(* Logix 5000 project; controller EuniceF_ICA14 vendor 1 type 14 code 150 rev 37.11; software revision 37.00 *)

TASK MainTask (continuous, watchdog 500 ms) : MainProgram

MODULES
   Local : vendor 1 type 14 code 150 (Compact 0, rev 37.11)
      Discrete_IO : Embedded (Compact 1, rev 3.1, Output RPI 20 ms)
      Analog_IO : Embedded (Compact 2, rev 1.1, Output RPI 80 ms)
      Counters : Embedded (Compact 3, rev 1.1, Output RPI 20 ms)
END_MODULES

VAR_GLOBAL   (* controller tags *)
   Button : BOOL;
   Light : BOOL;
   Seq1 : DINT;
   Timer1 : TIMER := (PRE := 2000);
END_VAR

PROGRAM MainProgram   (* main routine MainRoutine *)

ROUTINE MainRoutine   (* ladder *)
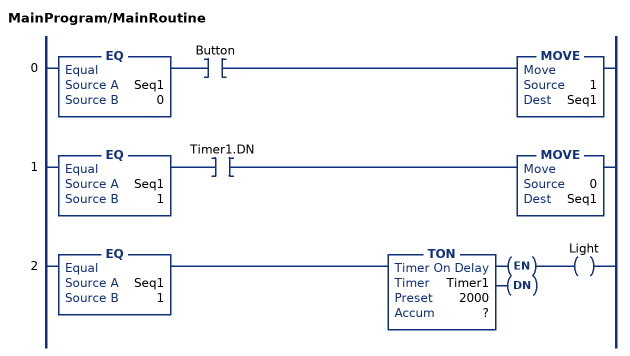
   0: EQ(Seq1,0)XIC(Button)MOVE(1,Seq1);
   1: EQ(Seq1,1)XIC(Timer1.DN)MOVE(0,Seq1);
   2: EQ(Seq1,1)TON(Timer1,?,?)OTE(Light);
END_ROUTINE
END_PROGRAM
